FUNCTION_BLOCK FB_Simple
VAR
	_bMember	: T_Bool := TRUE;
	_nMember 	: T_Dint := -57;
	_sMember 	: STRING := 'Testing Error.';
END_VAR

{attribute 'hide'}
METHOD FB_init : BOOL
VAR_INPUT
	bInitRetains : BOOL; // if TRUE, the retain variables are initialized (warm start / cold start)
	bInCopyCode : BOOL;  // if TRUE, the instance afterwards gets moved into the copy code (online change)
	bMember	: T_Bool;
	nMember : T_Dint;
	sMember : STRING;
END_VAR
THIS^._bMember := bMember;
THIS^._nMember := nMember;
THIS^._sMember := sMember;
END_METHOD

END_FUNCTION_BLOCK

(* stored: Version 1.1.0.1
   POU FB_Simple: Id {dc49e100-f1fa-47f6-a9fc-b3d52dc7fa87}, SpecialFunc None
   Method FB_init: Id {60f0206e-3a0d-4899-a0be-a72a6a95cd02} *)
